// TwinCAT 3 PLC project EE_Test_PLC_Code
// ProgramVersion: 3.1.4023.0
// libraries:
//   Tc2_Standard, * (Beckhoff Automation GmbH)
//   Tc2_System, * (Beckhoff Automation GmbH)
//   Tc3_Module, * (Beckhoff Automation GmbH)
// project tree:
//   JBOX_GVLs/ JBOX_GVL_IO.TcGVL
//   JBOX_POUs/ MAIN.TcPOU
//   / PlcTask.TcTTO
// real-time tasks:
//   TASK PlcTask: cycle T#10ms, priority 20, ADS port 350
// I/O:
//   DEVICE Device 1 (RT-Ethernet Adapter)
//   DEVICE Device 3 (EtherCAT), AmsNetId 10.14.30.245.4.1
//     Box 10 (CU2508) [CU2508 Ethernet Port]
//     C0 (EK1914) [EK1914, 2 Ch. Safety Input/Output 24V,  TwinSAFE]
//       modules: Module 1 (FSOE), Module 2 (DIO)
//       C1 (EL9410) [EL9410 E-Bus Power Supplier  (Diagnostics)]
//       C2 (EL2014) [EL2014 4Ch. Dig. Output 24V, 0,5A, Diagnostic]
//       C3 (EL1018) [EL1018 8Ch. Dig. Input 24V, 10µs]
//       C4 (EL1819) [EL1819 16Ch. Dig. Input 24V, 10µs]
//       C5 (EL1819) [EL1819 16Ch. Dig. Input 24V, 10µs]
//       C6 (EK1122-0008) [EK1122-0008 2 port EtherCAT junction M8]
//         B0 (EP9128-0021) [EP9128-0021 8x EtherCAT junction]
//           Term 19 (EK0000) [EK1100]
//           Term 20 (EP9128-1021) [EP9128-1021 8x EtherCAT junction - Dev A]
//           Term 21 (EP9128-2021) [EP9128-2021 8x EtherCAT junction - Dev B]
//     B1 (EP3184-0002) [EP3184-0002 4Ch. Ana. Input +/-10V, 0-10V, 0/4-20mA configurable, single ended]
//     B2 (EP1008-0002) [EP1008-0002 8 Ch. Dig. Input 24V, 3ms, M12]
//     B3 (EP3752-0000) [EP3752-0000 Acceleration Sensor]
//     B4 (EP1908) [EP1908, 8 Ch. Safety Input 24V, TwinSAFE ]
//       modules: Module 1 (FSOE)
//   DEVICE Device 4 (COM Port)
// variable links:
//   EE Test PLC Code/EE Test PLC Code Instance <-> Device 3 (EtherCAT)/B1 (EP3184-0002)
//     PlcTask Inputs/JBOX_GVL_IO.JB_PSU1_IOUT <-> AI Standard Channel 1/Value
//     PlcTask Inputs/JBOX_GVL_IO.JB_PSU2_IOUT <-> AI Standard Channel 2/Value
//   EE Test PLC Code/EE Test PLC Code Instance <-> Device 3 (EtherCAT)/B2 (EP1008-0002)
//     PlcTask Inputs/JBOX_GVL_IO.JB_DCDCS_OK <-> Channel 1/Input
//     PlcTask Inputs/JBOX_GVL_IO.JB_Door_Switch <-> Channel 4/Input
//     PlcTask Inputs/JBOX_GVL_IO.JB_PSUs_OK <-> Channel 2/Input
//   EE Test PLC Code/EE Test PLC Code Instance <-> Device 3 (EtherCAT)/C0 (EK1914)/C3 (EL1018)
//     PlcTask Inputs/JBOX_GVL_IO.J7_24V_Up <-> Channel 1/Input
//     PlcTask Inputs/JBOX_GVL_IO.J8_24V_Up <-> Channel 3/Input
//     PlcTask Inputs/JBOX_GVL_IO.J7_24V_Us <-> Channel 2/Input
//     PlcTask Inputs/JBOX_GVL_IO.J8_24V_Us <-> Channel 4/Input
//   EE Test PLC Code/EE Test PLC Code Instance <-> Device 3 (EtherCAT)/C0 (EK1914)/C4 (EL1819)
//     PlcTask Inputs/JBOX_GVL_IO.J{1..6}_24V_Up <-> Channel {1..11 step 2}/Input  (6 links)
//     PlcTask Inputs/JBOX_GVL_IO.J{1..6}_24V_Us <-> Channel {2..12 step 2}/Input  (6 links)
//   EE Test PLC Code/EE Test PLC Code Instance <-> Device 3 (EtherCAT)/C0 (EK1914)/C5 (EL1819)
//     PlcTask Inputs/JBOX_GVL_IO.SF1_MF_CONTINUITY <-> Channel 16/Input
//     PlcTask Inputs/JBOX_GVL_IO.SF2_MF_CONTINUITY <-> Channel 15/Input
//     PlcTask Inputs/JBOX_GVL_IO.SF4_Pull_Station <-> Channel 14/Input
//     PlcTask Inputs/JBOX_GVL_IO.SF6_MGT_CONTINUITY <-> Channel 13/Input
//     PlcTask Inputs/JBOX_GVL_IO.SF8_MGT_CONTINUITY <-> Channel 12/Input

CONFIGURATION EE_Test_PLC_Code
    RESOURCE PLC ON TwinCAT3
        TASK PlcTask(INTERVAL := T#10ms, PRIORITY := 20);
        PROGRAM MAIN WITH PlcTask : MAIN;
    END_RESOURCE
END_CONFIGURATION

// ---- JBOX_GVLs/JBOX_GVL_IO.TcGVL
{attribute 'qualified_only'}
VAR_GLOBAL

	
	
	// Boolean Variables linked to live data on ports
	{attribute 'TcLinkTo' := 'TIIB[C3 (EL1018)]^Channel 1^Input'}
	J7_24V_Up AT%I* : BOOL; //14.1 : BOOL; (*INDEX 4 24V PWR Check J7 (4) (1008 (1) port 2) *)
    {attribute 'TcLinkTo' := 'TIIB[C3 (EL1018)]^Channel 2^Input'}
	J7_24V_Us AT%I* : BOOL; //4.2 : BOOL; (*INDEX 5 24V PWR Check J7 (5) (1008 (1) port 3) *)    
	{attribute 'TcLinkTo' := 'TIIB[C3 (EL1018)]^Channel 3^Input'}
	J8_24V_Up AT%I* : BOOL; //5.4 : BOOL; (*INDEX 14 24V PWR Check J8 (4) (1008 (2) port 5) *)
    {attribute 'TcLinkTo' := 'TIIB[C3 (EL1018)]^Channel 4^Input'}
	J8_24V_Us AT%I* : BOOL; //5.5 : BOOL; (*INDEX 15 24V PWR Check J8 (5) (1008 (2) port 6) *)
	{attribute 'TcLinkTo' := 'TIIB[C4 (EL1819)]^Channel 1^Input'}	
	J1_24V_Up AT%I* : BOOL; //6.2 : BOOL; (*INDEX 20 Lighting 24V Check J1 (1) (1008 (3) port 3) *)
	{attribute 'TcLinkTo' := 'TIIB[C4 (EL1819)]^Channel 2^Input'}	
	J1_24V_Us AT%I* : BOOL; //6.3 : BOOL; (*INDEX 21 Lighting 24V Check J1 (2) (1008 (3) port 4) *)
	{attribute 'TcLinkTo' := 'TIIB[C4 (EL1819)]^Channel 3^Input'}	
	J2_24V_Up AT%I* : BOOL; //6.4 : BOOL; (*INDEX 22 Lighting 24V Check J2 (1) (1008 (3) port 5) *)
	{attribute 'TcLinkTo' := 'TIIB[C4 (EL1819)]^Channel 4^Input'}	
	J2_24V_Us AT%I* : BOOL; //6.5 : BOOL; (*INDEX 23 Lighting 24V Check J2 (2) (1008 (3) port 6) *)
	{attribute 'TcLinkTo' := 'TIIB[C4 (EL1819)]^Channel 5^Input'}	
	J3_24V_Up AT%I* : BOOL; //14.3 : BOOL; (*INDEX 6 24V PWR Check J3 (1) (1008 (1) port 4) *)
	{attribute 'TcLinkTo' := 'TIIB[C4 (EL1819)]^Channel 6^Input'}	
	J3_24V_Us AT%I* : BOOL; //4.4 : BOOL; (*INDEX 7 24V PWR Check J3 (2) (1008 (1) port 5) *)
	{attribute 'TcLinkTo' := 'TIIB[C4 (EL1819)]^Channel 7^Input'}	
	J4_24V_Up AT%I* : BOOL; //4.5 : BOOL; (*INDEX 8 24V PWR Check J4 (1) (1008 (1) port 6) *)
	{attribute 'TcLinkTo' := 'TIIB[C4 (EL1819)]^Channel 8^Input'}	
    J4_24V_Us AT%I* : BOOL; //4.7 : BOOL; (*INDEX 9 24V PWR Check J4 (2) (1008 (1) port 7) *)
	{attribute 'TcLinkTo' := 'TIIB[C4 (EL1819)]^Channel 9^Input'}	
	J5_24V_Up AT%I* : BOOL; //5.0 : BOOL; (*INDEX 10 24V PWR Check J5 (1) (1008 (2) port 1) *)
	{attribute 'TcLinkTo' := 'TIIB[C4 (EL1819)]^Channel 10^Input'}	
	J5_24V_Us AT%I* : BOOL; //5.1 : BOOL; (*INDEX 11 24V PWR Check J5 (2) (1008 (2) port 2) *)
	{attribute 'TcLinkTo' := 'TIIB[C4 (EL1819)]^Channel 11^Input'}	
	J6_24V_Up AT%I* : BOOL; //5.2 : BOOL; (*INDEX 12 24V PWR Check J6 (1) (1008 (2) port 3) *)
	{attribute 'TcLinkTo' := 'TIIB[C4 (EL1819)]^Channel 12^Input'}	
	J6_24V_Us AT%I* : BOOL; //5.3 : BOOL; (*INDEX 13 24V PWR Check J6 (2) (1008 (2) port 4) *)
	{attribute 'TcLinkTo' := 'TIIB[C5 (EL1819)]^Channel 16^Input'}	
	SF1_MF_CONTINUITY AT%I* : BOOL; //5.7 : BOOL; (*INDEX 17 Mine Phone Continuity SF1 (1008 (2) port 8) *)
	{attribute 'TcLinkTo' := 'TIIB[C5 (EL1819)]^Channel 15^Input'}	
	SF2_MF_CONTINUITY AT%I* : BOOL; //5.6 : BOOL; (*INDEX 16 Mine Phone Continuity SF2 (1008 (2) port 7) *)	
	{attribute 'TcLinkTo' := 'TIIB[C5 (EL1819)]^Channel 14^Input'}	
	SF4_Pull_Station AT%I* : BOOL; //4.0 : BOOL; (*INDEX 3 Fire pull Station SF4 (1008 (1) port 1) *)	
	{attribute 'TcLinkTo' := 'TIIB[C5 (EL1819)]^Channel 13^Input'}	
	SF6_MGT_CONTINUITY AT%I* : BOOL; //6.0 : BOOL; (*INDEX 18 MGT Continuity SF6 (1008 (3) port 1) *)
	{attribute 'TcLinkTo' := 'TIIB[C5 (EL1819)]^Channel 12^Input'}	
	SF8_MGT_CONTINUITY AT%I* : BOOL; //6.1: BOOL; (*INDEX 19 MGT Continuity SF8 (1008 (3) port 2) *)
	
	
	{attribute 'TcLinkTo' := 'TIIB[B2 (EP1008-0002)]^Channel 4^Input'}
	JB_Door_Switch AT%I* : BOOL; (* Door Switch *)
	{attribute 'TcLinkTo' := 'TIIB[B2 (EP1008-0002)]^Channel 1^Input'}
	JB_DCDCS_OK AT%I* : BOOL; (* JBOX DCDC GOOD Signal *)
	{attribute 'TcLinkTo' := 'TIIB[B2 (EP1008-0002)]^Channel 2^Input'}
	JB_PSUs_OK AT%I* : BOOL; (* PSUs OK *)
	//{attribute 'TcLinkTo' := 'TIIB[C2 (EL2014)]^DIG Outputs^Channel 2^Output'}
	//SF5_Fire_Alarm AT%Q* : BOOL; //3.1 : BOOL; (*INDEX 0 Fire Alarm Sound SF5 (2024 port 2) *)
	{attribute 'TcLinkTo' := 'TIIB[B1 (EP3184-0002)]^AI Standard Channel 1^Value'}
	JB_PSU1_IOUT AT%I* : INT; 
	{attribute 'TcLinkTo' := 'TIIB[B1 (EP3184-0002)]^AI Standard Channel 2^Value'}
	JB_PSU2_IOUT AT%I* : INT;
	
	
END_VAR

// ---- JBOX_POUs/MAIN.TcPOU
PROGRAM MAIN
VAR_INPUT
END_VAR
VAR
END_VAR

END_PROGRAM
